// TIA Portal V19 export
VAR_GLOBAL   // PLC tag table "Peeler_IO"
   Peeler_V_Bwd AT %Q103.5 : Bool;   // 810YV3
   Peeler_V_Fwd AT %Q103.6 : Bool;   // 810YV4
   Peeler_Ls_Bwd AT %I129.3 : Bool;   // 810SQ3
   Peeler_V_Down AT %Q103.4 : Bool;   // 810YV2
   Peeler_V_Up AT %Q103.3 : Bool;   // 810YV1
   Peeler_Ls_Down AT %I129.2 : Bool;   // 810SQ2
   Peeler_Ls_Fwd AT %I129.4 : Bool;   // 810SQ4
   Peeler_Ls_Up AT %I129.1 : Bool;   // 810SQ1
END_VAR
